{attribute 'qualified_only'}
{attribute 'strict'}
TYPE E_Manufacturer :
(
	Unknown_manufacturer := 0,
	Hengstler
);
END_TYPE

(* stored: Version 1.1.0.1, ProductVersion 3.1.4024.12
   DUT E_Manufacturer: Id {2f3d39fb-e187-4571-a5c4-f4d699bd41d2} *)
